// TIA Portal V16 export
// export: Created 2022-07-21T09:35:31.7102223Z, ExportSetting WithDefaults, DisplayName Totally Integrated Automation Portal, DisplayVersion V16 Update 4, DisplayName TIA Portal Version Control Interface, DisplayVersion V16 Update 2, DisplayName TIA Portal Openness, DisplayVersion V16 Update 4, DisplayName SINAMICS Startdrive Advanced, DisplayVersion V16 Update 5, DisplayName SINAMICS Startdrive G130, G150, S120, S150, SINAMICS MV, S210, DisplayVersion V16 Update 5, DisplayName SINAMICS Startdrive G110M, G120, G120C, G120D, G120P, G115D, DisplayVersion V16 Update 5, DisplayName STEP 7 Professional, DisplayVersion V16 Update 4, DisplayName STEP 7 Safety, DisplayVersion V16, DisplayName WinCC Advanced, DisplayVersion V16 Update 4
FUNCTION_BLOCK "fbCycleTime"   // FB4, LAD
TITLE = Cycle time / Czas cyklu
{ S7_Optimized_Access := 'TRUE' }
VERSION : 0.1
// stored: AutoNumber true, IsIECCheckEnabled true, IsRetainMemResEnabled false, MemoryReserve 100, SetENOAutomatically false, UDAEnableTagReadback false
   VAR_INPUT
      InitialCall { ExternalAccessible := 'False'; ExternalVisible := 'False'; ExternalWritable := 'False'} : Bool;
   END_VAR
   VAR
      sRuntimeMemory { ExternalAccessible := 'False'; ExternalVisible := 'False'; ExternalWritable := 'False'} : LReal;   // Gespeicherte Zeit für Funktion Runtime, darf nicht remanent sein / Saved time for function Runtime, must be non-retain
      sRestMilliseconds { ExternalAccessible := 'False'; ExternalVisible := 'False'; ExternalWritable := 'False'} : LReal;   // Restwert für Millisekunden / Rest value for milliseconds
      sRestMicroseconds { ExternalAccessible := 'False'; ExternalVisible := 'False'; ExternalWritable := 'False'} : LReal;   // Restwert für Mikrosekunden / Rest value for microseconds
      tCurrentRuntime { ExternalAccessible := 'False'; ExternalVisible := 'False'; ExternalWritable := 'False'} : LReal;   // Letzte Zykluszeit in Sekunden / Previous scantime in seconds
   END_VAR
   VAR_TEMP
      tRuntimeMilliseconds : LReal;   // Letzte Zykluszeit in Millisekunden / Previous scantime in milliseconds
      tRuntimeMicroseconds : LReal;   // Letzte Zykluszeit in Mikrosekunden / Previous scantime in microseconds
   END_VAR
BEGIN

REGION Network 1: Current cycle time / Aktualny czas cyklu
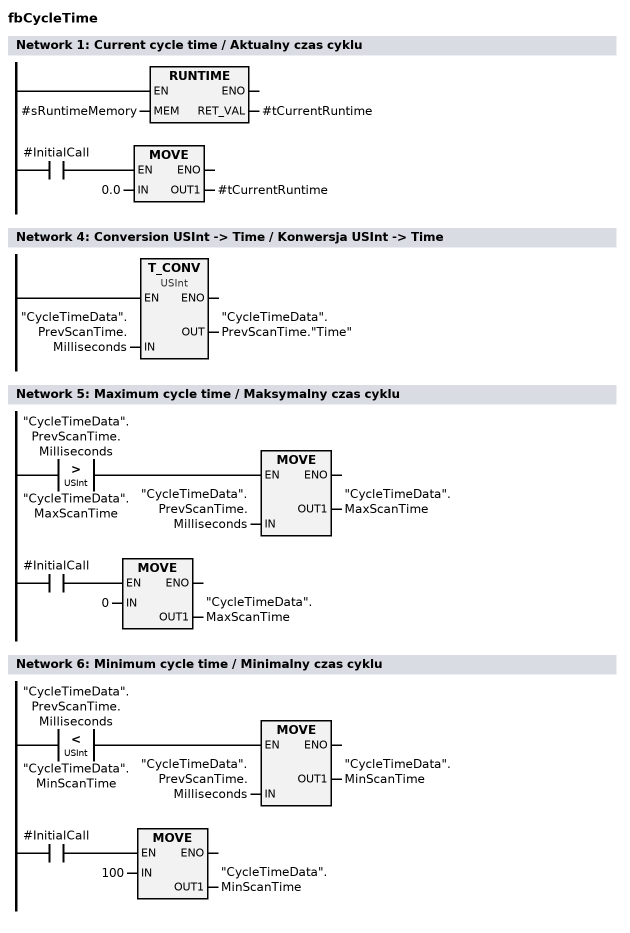
   // no SCL statement known for Runtime: written as a call
   #tCurrentRuntime := Runtime(mem := #sRuntimeMemory);
   IF #InitialCall THEN #tCurrentRuntime := 0.0; END_IF;
END_REGION

REGION Network 2 (SCL): Previous cycle time [ms] / Czas poprzedniego cyklu [ms]
   //-- Dodanie resztu ostatniego runtime do obecnego runtime
   #tRuntimeMilliseconds := (#tCurrentRuntime * 1000.0) + #sRestMilliseconds;

   //-- Zapis do DB
   "CycleTimeData".PrevScanTime.Milliseconds := FLOOR_USINT(IN := #tRuntimeMilliseconds);

   //-- Zapis reszty runtime dla następnego cyklu
   #sRestMilliseconds := #tRuntimeMilliseconds - "CycleTimeData".PrevScanTime.Milliseconds;
END_REGION

REGION Network 3 (SCL): Previous cycle time [us] / Czas poprzedniego cyklu [us]
   //-- Dodanie resztu ostatniego runtime do obecnego runtime
   #tRuntimeMicroseconds := (#tCurrentRuntime * 1000000.0) + #sRestMicroseconds;

   //-- Zapis do DB
   "CycleTimeData".PrevScanTime.Microseconds := FLOOR_UINT(IN := #tRuntimeMicroseconds);

   //-- Zapis reszty runtime dla następnego cyklu
   #sRestMicroseconds := #tRuntimeMicroseconds - "CycleTimeData".PrevScanTime.Microseconds;
END_REGION

REGION Network 4: Conversion USInt -> Time / Konwersja USInt -> Time
   RUNG wire#powerrail
      { S7_Templates := "[src_type := USInt, dest_type := Time]" } T_CONV(IN := "CycleTimeData".PrevScanTime.Milliseconds, OUT => "CycleTimeData".PrevScanTime."Time")
   END_RUNG
   // the same network as SCL:
   T_CONV(IN := "CycleTimeData".PrevScanTime.Milliseconds, OUT => "CycleTimeData".PrevScanTime."Time");
END_REGION

REGION Network 5: Maximum cycle time / Maksymalny czas cyklu
   RUNG wire#powerrail
      { S7_Templates := "SrcType := USInt" } GT_Contact(in1 := "CycleTimeData".PrevScanTime.Milliseconds, in2 := "CycleTimeData".MaxScanTime)
      Move(in := "CycleTimeData".PrevScanTime.Milliseconds, out1 => "CycleTimeData".MaxScanTime)
   END_RUNG
   RUNG wire#powerrail
      Contact( #InitialCall )
      Move(in := 0, out1 => "CycleTimeData".MaxScanTime)
   END_RUNG
   // the same network as SCL:
   IF "CycleTimeData".PrevScanTime.Milliseconds > "CycleTimeData".MaxScanTime THEN
       "CycleTimeData".MaxScanTime := "CycleTimeData".PrevScanTime.Milliseconds;
   END_IF;
   IF #InitialCall THEN "CycleTimeData".MaxScanTime := 0; END_IF;
END_REGION

REGION Network 6: Minimum cycle time / Minimalny czas cyklu
   RUNG wire#powerrail
      { S7_Templates := "SrcType := USInt" } LT_Contact(in1 := "CycleTimeData".PrevScanTime.Milliseconds, in2 := "CycleTimeData".MinScanTime)
      Move(in := "CycleTimeData".PrevScanTime.Milliseconds, out1 => "CycleTimeData".MinScanTime)
   END_RUNG
   RUNG wire#powerrail
      Contact( #InitialCall )
      Move(in := 100, out1 => "CycleTimeData".MinScanTime)
   END_RUNG
   // the same network as SCL:
   IF "CycleTimeData".PrevScanTime.Milliseconds < "CycleTimeData".MinScanTime THEN
       "CycleTimeData".MinScanTime := "CycleTimeData".PrevScanTime.Milliseconds;
   END_IF;
   IF #InitialCall THEN "CycleTimeData".MinScanTime := 100; END_IF;
END_REGION
END_FUNCTION_BLOCK
